# EPICS autosave request: support/pilatus/1-6/pilatusApp/Db/pilatusROI_settings.req
$(DET)AcquireMode
$(DET)ExposureTime
$(DET)NImages
$(DET)ExposurePeriod
$(DET)NExposures
$(DET)DelayTime
$(DET)FilePath
$(DET)Filename
$(DET)FileFormat
$(DET)FileNumber
$(DET)AutoIncrement
$(DET)BadPixelFile
$(DET)FlatFieldFile
$(DET)MinFlatField
$(DET)ThresholdEnergy
$(DET)Gain
$(DET)ReadTiffTimeout
$(DET)MinWFUpdateTime
$(DET)PostImages
$(DET)HighlightROIs
$(DET)MinImageUpdateTime
